RoboDK station: Kuka_RoboDK.rdk

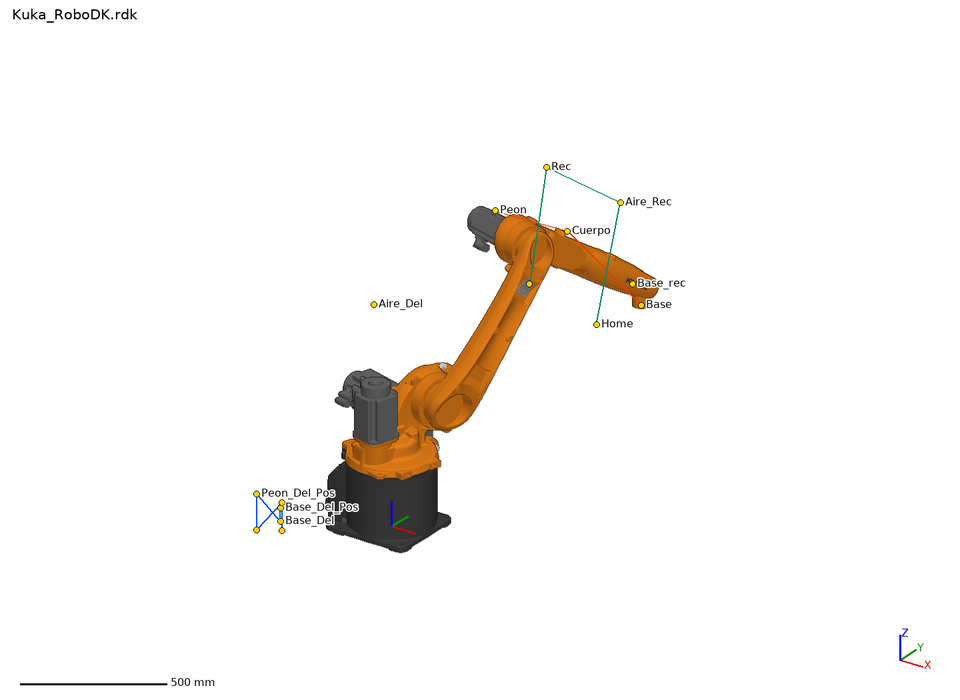
[picture v0: the station drawn from its stored meshes, robots at their saved joint values, targets as dots, program paths as lines]
Station Kuka_Prueba (saved by RoboDK 5.6.3). Poses are relative to the parent item; angles as X-Y-Z fixed-axis rotations.
Station parameters (name, value as stored): IO_5, 1
  - Python program Programa para analisis de movimiento de aire (listed below)
  - Python program Programa para parte de arriba (listed below)
  - Python program Prueba movimientos (listed below)
  - frame KUKA KR 10 R1420 Base at (0, 0, 0) mm
    - robot KUKA KR 10 R1420: 6 axes, payload 10 kg, reach 1420 mm, repeatability 0.04 mm, weight 160 kg
        modified DH rows (alpha deg, a mm, theta deg, d mm): 0, 0, 0, 450; -90, 150, 0, 0; 0, 610, -90, 0; -90, 20, 0, 660; 90, 0, 0, 0; -90, 0, 180, 80
        joint limits [-170, -185, -137, -185, -120, -350] to [170, 65, 163, 185, 120, 350]; home [0, -90, 90, 0, 0, 0]; saved at [-74.055, -51.44, 84.878, 0, 56.562, 18.445]
      - tool Tool 1, TCP at (0, 0, 0) mm
    - target Home (Cartesian target) at (850, 0, 1000) mm, rotated rx 180 ry 0 rz -180 deg; joints [0, -86.236, 86.122, 0, 90.114, 0] of KUKA KR 10 R1420
    - target Aire_Del (Cartesian target) at (467.8, -773.44, 1278.03) mm, rotated rx -179.59 ry 64.82 rz 130.84 deg; joints [59.632, -83.021, 61.89, -12.366, 47.324, 12.946] of KUKA KR 10 R1420
    - target Aire_Rec (Cartesian target) at (549.78, 569.9, 1149.03) mm, rotated rx 180 ry 0 rz -134.9 deg; joints [-46.029, -89.666, 76.568, 0, 103.098, -0.928] of KUKA KR 10 R1420
    - target Rec (Cartesian target) at (12, 900, 1000) mm, rotated rx 178.8 ry 0 rz -90 deg; joints [-89.129, -81.483, 80.901, -1.204, 90.601, 0.858] of KUKA KR 10 R1420
    - target Base (Cartesian target) at (300, 1050, 500) mm, rotated rx 180 ry 0 rz -87.5 deg; joints [-74.055, -51.44, 84.878, 0, 56.562, 18.445] of KUKA KR 10 R1420
    - target Base_rec (Cartesian target) at (300, 1000, 600) mm, rotated rx 180 ry 0 rz -87.5 deg; joints [-73.301, -60.005, 88.598, 0, 61.407, 19.199] of KUKA KR 10 R1420
    - target Base_Del (Cartesian target) at (138, -855, 400) mm, rotated rx 180 ry 0 rz -180 deg; joints [80.831, -61.444, 113.175, 0, 38.268, 80.831] of KUKA KR 10 R1420
    - target Base_Del_Pos (Cartesian target) at (138, -855, 450) mm, rotated rx 180 ry 0 rz -180 deg; joints [80.831, -65.183, 112.756, 0, 42.428, 80.831] of KUKA KR 10 R1420
    - target Cuerpo (Cartesian target) at (1, 1040, 700) mm, rotated rx 180 ry 0 rz -88.5 deg; joints [-89.945, -64.053, 85.113, 0, 68.939, 1.555] of KUKA KR 10 R1420
    - target Cuerpo_Del (Cartesian target) at (36.5, -699, 275) mm, rotated rx 0 ry 90 rz -90 deg; joints [86.625, -51.719, 135.431, -3.395, -83.723, 0.372] of KUKA KR 10 R1420
    - target Cuerpo_Del_Pos (Cartesian target) at (36.5, -699, 380) mm, rotated rx 0 ry 90 rz -90 deg; joints [86.625, -65.309, 138.018, -3.534, -72.74, 1.05] of KUKA KR 10 R1420
    - target Peon (Cartesian target) at (-290.5, 1028, 700) mm, rotated rx 180 ry 0 rz -88.5 deg; joints [-105.78, -61.512, 81.439, 0, 70.073, -14.28] of KUKA KR 10 R1420
    - target Peon_Del (Cartesian target) at (-71.7, -695, 245) mm, rotated rx 0 ry 90 rz -90 deg; joints [96.65, -47.893, 134.402, 6.662, -86.532, -0.405] of KUKA KR 10 R1420
    - target Peon_Del_Pos (Cartesian target) at (-71.7, -695, 380) mm, rotated rx 0 ry 90 rz -90 deg; joints [96.65, -65.349, 138.106, 6.96, -72.877, -2.058] of KUKA KR 10 R1420
    - target Ruta aerea inferior (Cartesian target) at (12, 800, 600) mm, rotated rx 178.8 ry 0 rz -90 deg; joints [-89.02, -80.188, 116.118, -1.486, 54.099, 1.852] of KUKA KR 10 R1420
  - program Posiciones_Del (7 instructions, listed below)
  - program Posiciones_Rec (4 instructions, listed below)
  - program Prog9 (2 instructions, listed below)
  - program Ruta inferior (5 instructions, listed below)
  - program Prueba 1 (4 instructions, listed below)
  - Python program Prueba principal (listed below)
  - Python program gripper (listed below)
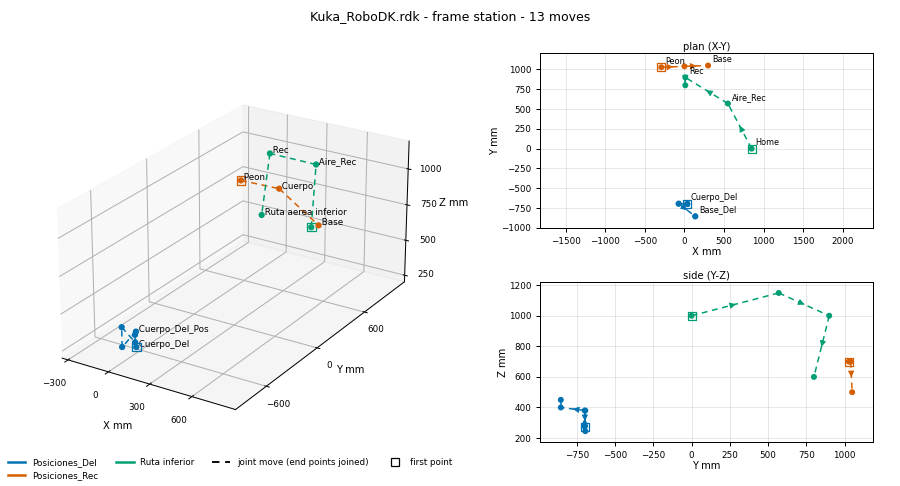
[picture p0: tool path of Kuka_RoboDK.rdk in frame station, 13 of 13 moves have a stored position in this frame; points joined in program order, loops and branches not executed]

--- Python program Programa para analisis de movimiento de aire ---
# Librerias
from robolink import *
from robodk import *

# Inicializacion de robo DK
RL = Robolink()

# Guardado de localizaciones para objetivos en variables
robot = RL.Item('KUKA KR 10 R1420')
home = RL.Item('Home')
peon = RL.Item('Peon')
cuerpo = RL.Item('Cuerpo')
base = RL.Item('Base')
Rec = RL.Item('Rec')
ARec = RL.Item('Aire_Rec')
ADel = RL.Item('Aire_Del')
cuerpodelpos = RL.Item('Cuerpo_Del_Pos')
cuerpodel = RL.Item('Cuerpo_Del')
peondelpos = RL.Item('Peon_Del_Pos')
peondel = RL.Item('Peon_Del')
basedelpos = RL.Item('Base_Del_Pos')
basedel = RL.Item('Base_Del')
rutainf = RL.Item('Ruta aerea inferior')

# Movimientos a hacer (se hizo una doble ejecucion para evitar saltos en el el programa que se traba algunas veces)
# Movimientos de Peon ##################################################

robot.setSpeed(130)
robot.MoveJ(home)
robot.MoveJ(home)
robot.MoveJ(ARec)
robot.MoveJ(ARec)
robot.MoveJ(Rec)
robot.MoveJ(Rec)
robot.MoveJ(ADel)
robot.MoveJ(ADel)
robot.MoveJ(home)
robot.MoveJ(home)

--- Python program Programa para parte de arriba ---
# Librerias
from robolink import *
from robodk import *

# Inicializacion de robo DK
RL = Robolink()

# Guardado de localizaciones para objetivos en variables
robot = RL.Item('KUKA KR 10 R1420')
home = RL.Item('Home')
peon = RL.Item('Peon')
cuerpo = RL.Item('Cuerpo')
base = RL.Item('Base')
Rec = RL.Item('Rec')
ARec = RL.Item('Aire_Rec')
ADel = RL.Item('Aire_Del')
cuerpodelpos = RL.Item('Cuerpo_Del_Pos')
cuerpodel = RL.Item('Cuerpo_Del')
peondelpos = RL.Item('Peon_Del_Pos')
peondel = RL.Item('Peon_Del')
basedelpos = RL.Item('Base_Del_Pos')
basedel = RL.Item('Base_Del')
rutainf = RL.Item('Ruta aerea inferior')

# Movimientos a hacer (se hizo una doble ejecucion para evitar saltos en el el programa que se traba algunas veces)
# Movimientos de Peon ##################################################

robot.setSpeed(250)
robot.MoveJ(home)
robot.MoveJ(home)
robot.MoveJ(ARec)
robot.MoveJ(ARec)
robot.MoveJ(Rec)
robot.MoveJ(Rec)
robot.setSpeed(150)
robot.MoveJ(peon)
robot.MoveJ(peon)
robot.MoveJ(Rec)
robot.MoveJ(Rec)
robot.setSpeed(230)
robot.MoveJ(ARec)
robot.MoveJ(ARec)
robot.MoveJ(home)
robot.MoveJ(home)
robot.MoveJ(ADel)
robot.MoveJ(ADel)
robot.setSpeed(150)
robot.MoveJ(peondelpos)
robot.MoveJ(peondelpos)
robot.MoveJ(ADel)
robot.MoveJ(ADel)
robot.setSpeed(230)
robot.MoveJ(home)
robot.MoveJ(home)

--- Python program Prueba movimientos ---
# Librerias
from robolink import *
from robodk import *

# Inicializacion de robo DK
RL = Robolink()

# Guardado de localizaciones para objetivos en variables
robot = RL.Item('KUKA KR 10 R1420')
home = RL.Item('Home')
peon = RL.Item('Peon')
cuerpo = RL.Item('Cuerpo')
base = RL.Item('Base')
Rec = RL.Item('Rec')
ARec = RL.Item('Aire_Rec')
ADel = RL.Item('Aire_Del')
cuerpodelpos = RL.Item('Cuerpo_Del_Pos')
cuerpodel = RL.Item('Cuerpo_Del')
peondelpos = RL.Item('Peon_Del_Pos')
peondel = RL.Item('Peon_Del')
basedelpos = RL.Item('Base_Del_Pos')
basedel = RL.Item('Base_Del')
rutainf = RL.Item('Ruta aerea inferior')

# Movimientos a hacer (se hizo una doble ejecucion para evitar saltos en el el programa que se traba algunas veces)
# Movimientos de Peon ##################################################
robot.setSpeed(250)
robot.MoveJ(home)
robot.MoveJ(home)
robot.MoveJ(ARec)
robot.MoveJ(ARec)
robot.MoveJ(Rec)
robot.MoveJ(Rec)
robot.setSpeed(150)
robot.MoveJ(base)
robot.MoveJ(base)
robot.MoveJ(Rec)
robot.MoveJ(Rec)
robot.setSpeed(230)
robot.MoveJ(ARec)
robot.MoveJ(ARec)
robot.MoveJ(home)
robot.MoveJ(home)
robot.MoveJ(ADel)
robot.MoveJ(ADel)
robot.setSpeed(150)
robot.MoveJ(basedelpos)
robot.MoveJ(basedelpos)
robot.MoveJ(ADel)
robot.MoveJ(ADel)
robot.setSpeed(230)
robot.MoveJ(home)
robot.MoveJ(home)

--- program Posiciones_Del (robot KUKA KR 10 R1420) ---
  Est. Ref.: KUKA KR 10 R1420 Base
  MoveJ (Cuerpo_Del)
  MoveJ (Cuerpo_Del_Pos)
  MoveJ (Peon_Del)
  MoveJ (Peon_Del_Pos)
  MoveJ (Base_Del)
  MoveJ (Base_Del_Pos)

--- program Posiciones_Rec (robot KUKA KR 10 R1420) ---
  Est. Ref.: KUKA KR 10 R1420 Base
  MoveJ (Peon)
  MoveJ (Cuerpo)
  MoveJ (Base)

--- program Prog9 (robot KUKA KR 10 R1420) ---
  Set IO_5=1
  Set IO_5=1

--- program Ruta inferior (robot KUKA KR 10 R1420) ---
  Set Ref.: KUKA KR 10 R1420 Base
  MoveJ (Home)
  MoveJ (Aire_Rec)
  MoveJ (Rec)
  MoveJ (Ruta aerea inferior)

--- program Prueba 1 (robot KUKA KR 10 R1420) ---
  Est. Ref.: KUKA KR 10 R1420 Base
  Establecer velocidad (230.0 mm/s)
  Llamar Prueba 1(1)
  Set IO_5=1

--- Python program Prueba principal ---
# Librerias
from robolink import *
from robodk import *
#import robotiqGripper as rq
import serial
import time
import binascii

# Inicializacion de robo DK
RL = Robolink()

# Guardado de localizaciones para objetivos en variables
robot = RL.Item('KUKA KR 10 R1420')
home = RL.Item('Home')
peon = RL.Item('Peon')
cuerpo = RL.Item('Cuerpo')
base = RL.Item('Base')
Rec = RL.Item('Rec')
ARec = RL.Item('Aire_Rec')
ADel = RL.Item('Aire_Del')
cuerpodelpos = RL.Item('Cuerpo_Del_Pos')
cuerpodel = RL.Item('Cuerpo_Del')
peondelpos = RL.Item('Peon_Del_Pos')
peondel = RL.Item('Peon_Del')
basedelpos = RL.Item('Base_Del_Pos')
basedel = RL.Item('Base_Del')
rutainf = RL.Item('Ruta aerea inferior')

# Movimientos a hacer (se hizo una doble ejecucion para evitar saltos en el el programa que se traba algunas veces)
# Movimientos de Peon ##################################################
robot.setSpeed(250)
robot.MoveJ(home)
robot.MoveJ(home)
robot.MoveJ(ARec)
robot.MoveJ(ARec)
robot.MoveJ(Rec)
robot.MoveJ(Rec)
robot.setSpeed(100)
robot.MoveJ(base)
robot.MoveJ(base)


# Configuración de la conexión serial para el gripper (ajusta según tu configuración)
ser = serial.Serial(port='/dev/ttyUSB0', baudrate=115200, timeout=1,
parity=serial.PARITY_NONE, stopbits=serial.STOPBITS_ONE, bytesize=serial.EIGHTBITS)

# Función para enviar comandos Modbus RTU al gripper
def send_modbus_command(register, value):
    command = bytearray([9, 16, (register >> 8) & 0xFF, register & 0xFF,
                         0, 6, 12, 3, 0, 0, (value >> 8) & 0xFF, value & 0xFF,
                         0, 0, 0, 0])
    crc = binascii.crc32(command) & 0xFFFF
    command.append((crc >> 8) & 0xFF)
    command.append(crc & 0xFF)
    ser.write(command)

# Esperar un tiempo para que el robot alcance la posición (ajusta según tus necesidades)
time.sleep(4)

# Enviar el comando para cerrar el gripper
send_modbus_command(1000, 1)  # Ajusta la dirección del registro según tu configuración

# Esperar un tiempo para que el gripper se cierre (ajusta según tus necesidades)
time.sleep(2)




# Obtener la matriz de transformación actual del objetivo
current_pose = robot.Pose()

# Definir el nuevo ángulo de rotación en el eje Z en grados (por ejemplo, 45 grados)
new_rotation_angle_degrees = 45

# Convertir el ángulo de grados a radianes
new_rotation_angle_radians = math.radians(new_rotation_angle_degrees)

# Calcular la nueva matriz de transformación con la rotación en el eje Z
rotation_matrix_z = Mat([
    [math.cos(new_rotation_angle_radians), -math.sin(new_rotation_angle_radians), 0, 0],
    [math.sin(new_rotation_angle_radians), math.cos(new_rotation_angle_radians), 0, 0],
    [0, 0, 1, 0],
    [0, 0, 0, 1]
])

# Combinar la nueva rotación con la matriz de transformación actual
new_pose = current_pose * rotation_matrix_z

# Actualizar la posición del objetivo con la nueva rotación
robot.MoveJ(new_pose)

# Obtener la cantidad en la que deseas cambiar el eje Z
desplazamiento_z = -200  # Cambia esta cantidad según tus necesidades

# Obtener la matriz de transformación actual del robot
current_pose = robot.Pose()

# Crear una nueva matriz de translación en el eje Z
new_translacion_z = transl(0, 0, desplazamiento_z)

# Combinar la nueva translación con la matriz de transformación actual
new_pose = current_pose * new_translacion_z

# Aplicar la nueva posición al robot
robot.MoveJ(new_pose)

robot.MoveJ(Rec)
robot.MoveJ(Rec)
robot.MoveJ(ARec)
robot.MoveJ(ARec)
robot.MoveJ(home)
robot.MoveJ(home)
robot.MoveJ(ADel)
robot.MoveJ(ADel)
robot.MoveJ(basedel)
robot.MoveJ(basedel)

# Esperar un tiempo para que el gripper se abra (ajusta según tus necesidades)
time.sleep(4)

# Enviar el comando para abrir el gripper
send_modbus_command(1000, 0)  # Ajusta la dirección del registro según tu configuración

# Esperar un tiempo para que el gripper se abra (ajusta según tus necesidades)
time.sleep(2)

robot.MoveJ(ADel)
robot.MoveJ(ADel)
robot.MoveJ(home)
robot.MoveJ(home)

--- Python program gripper ---
import minimalmodbus
import serial
import binascii
import time
import robotiqGripper as rq

instrument = minimalmodbus.Instrument('COM5', 9, debug = True)

# instrument.serial.port                     # this is the serial port name
instrument.serial.baudrate = 115200         # Baud
# instrument.serial.bytesize = 8
# instrument.serial.parity   = serial.PARITY_NONE
# instrument.serial.stopbits = 1
# instrument.serial.timeout  = 0.2          # seconds
# instrument.address = 9                         # this is the slave address number
# instrument.mode = minimalmodbus.MODE_RTU   # rtu or ascii mode
# instrument.clear_buffers_before_each_transaction = True
#
# print(instrument)

# instrument.write_registers(1000,[0,0,0]) # Reset the gripper
# instrument.write_registers(1000,[256,0,0]) #Activate the gripper


myGripper = rq.RobotiqGripper(portname='COM5',slaveaddress=9)
myGripper.activate()
myGripper.openGripper(1,1)
myGripper.closeGripper(1,1)
time.sleep(5)
myGripper.openGripper(255,255)
myGripper.closeGripper(255,255)
time.sleep(2)
myGripper.goTo(0)
time.sleep(1)
myGripper.goTo(125)
time.sleep(1)
myGripper.goTo(255)
time.sleep(2)
myGripper.goTo(0)
